{attribute 'linkalways'} 
{attribute 'no_explicit_call' := 'This FB is a CLASS and must be accessed using methods or properties'}
{attribute 'enable_dynamic_creation'}
FUNCTION_BLOCK AsyncServerResponse IMPLEMENTS I_ServerResponse
VAR
	serverResponse : I_ServerResponse;
	asyncResponseManager : I_AsyncResponseManager;
END_VAR

METHOD PUBLIC Accepted
VAR_INPUT
END_VAR
serverResponse.Accepted();
END_METHOD

METHOD PUBLIC Busy
VAR_INPUT
END_VAR
serverResponse.Busy();
END_METHOD

METHOD PUBLIC Error
VAR_INPUT
	Message : T_MAXSTRING;
END_VAR
serverResponse.Error(Message);
END_METHOD

METHOD FB_init : BOOL
VAR_INPUT
	bInitRetains : BOOL; // if TRUE, the retain variables are initialized (warm start / cold start)
	bInCopyCode : BOOL;  // if TRUE, the instance afterwards gets moved into the copy code (online change)
	ServerResponse : I_ServerResponse;
	AsyncResponseManager : I_AsyncResponseManager;
END_VAR
THIS^.serverResponse := ServerResponse;
This^.asyncResponseManager := AsyncResponseManager;
END_METHOD

PROPERTY PUBLIC Header : I_Header
GET
Header := serverResponse.Header;
END_GET
END_PROPERTY

PROPERTY PUBLIC HeadersSent : BOOL
GET
HeadersSent := serverResponse.HeadersSent;
END_GET
END_PROPERTY

METHOD PUBLIC Pending
VAR_INPUT
	ResponseId : REFERENCE TO T_MAXSTRING;
	RetryDelayInMs : UDINT;
END_VAR
asyncResponseManager.HandlePending(serverResponse, ResponseId, RetryDelayInMs);
END_METHOD

METHOD PUBLIC Success
VAR_INPUT
END_VAR
serverResponse.Success();
END_METHOD

METHOD PUBLIC SuccessWithPayload
VAR_INPUT
	PayloadDataAddress : PVOID;
	PayloadDataSize : UDINT;
END_VAR
serverResponse.SuccessWithPayload(PayloadDataAddress, PayloadDataSize);
END_METHOD

END_FUNCTION_BLOCK

(* stored: Version 1.1.0.1, ProductVersion 3.1.4024.12
   POU AsyncServerResponse: Id {5279022d-433f-46df-8aa0-20f3d6e3dc4e}, SpecialFunc None
   Folder Constructor: Id {7472a293-bc0b-4d28-919f-6f4387813456}
   Method Accepted: Id {3f6f7ea2-6994-4c3d-9c41-d9f8236b0d04}
   Method Busy: Id {b7ecd058-1eb0-4675-98a2-e0ab00a0924d}
   Method Error: Id {b26c2977-852c-4f2a-b9c9-fc3e67f7242a}
   Method FB_init: Id {98d80c83-8412-4837-90cf-d15291aa0120}
   Property Header: Id {f9f8c5b5-0cd5-4f19-bebb-b3678d4adb6f}
   Get Get: Id {82cbb266-0398-4ec0-a13e-b03276a2b0c4}
   Property HeadersSent: Id {802f509f-a21c-492d-b35c-183d9d69898a}
   Get Get: Id {5b5e6204-b5ca-42ca-9bb3-c73446a49942}
   Method Pending: Id {8f6fae18-499a-4115-809e-b02e280e4409}
   Method Success: Id {edd54756-c1d6-45d4-8aed-a5f86d7181cf}
   Method SuccessWithPayload: Id {4cf9b931-834b-420d-9f2d-3690e7fb763a} *)
